(* IEC 61131-3 sources: ics/BLR1_PhoenixContact/BLR1_AXC1050_21/LogicalPOUs/VLV, 3 files *)

(* ---- ValveFB.ST ---- *)
(*@PROPERTIES_EX@
TYPE: POU
LOCALE: 0
IEC_LANGUAGE: ST
PLC_TYPE: independent
PROC_TYPE: independent
GROUP: VLVS.FB
*)
(*@KEY@:DESCRIPTION*)

(*@KEY@:END_DESCRIPTION*)
FUNCTION_BLOCK ValveFB

(*Group:Default*)

VAR
    Fb_Alrm_Tmr :    TON;
END_VAR

VAR_IN_OUT
    Vlv_strct :    VLV;
    Aux_strct :    VLV_MISC;
END_VAR

VAR
    AlrmNotMove :    BOOL;
    AlrmSQ :    BOOL;
    RunManual :    BOOL;
    RunAuto :    BOOL;
    COM_Open :    BOOL;
    COM_Close :    BOOL;
END_VAR

VAR_INPUT
    Cycle :    CCL;
END_VAR

VAR
    NotMove_Alrm_Tmr :    TON;
    AlrmFeedBack :    BOOL;
    AlarmBlock :    BOOL;
END_VAR

VAR_EXTERNAL
    TICK_1S_PLS :    BOOL;
END_VAR

(*@KEY@: WORKSHEET
NAME: ValveFB
IEC_LANGUAGE: ST
*)

IF TICK_1S_PLS and not Aux_strct.AuxFlag THEN
    Aux_strct.Tick_1S:= TRUE;
END_IF;
Aux_strct.AuxFlag:= TICK_1S_PLS;

(*============================================================================*)
    (*Alarm Feedback processing*)
(*============================================================================*)
IF Vlv_strct.CW.Enable and (Aux_strct.COM_Close or Aux_strct.COM_Open) and
    not Vlv_strct.SW.RUN THEN
    IF Aux_strct.Tick_1S THEN
        Aux_strct.FbAlarmTickCount:= Aux_strct.FbAlarmTickCount + 1;
    END_IF;
ELSE
    Aux_strct.FbAlarmTickCount:= 0;
END_IF;

IF Vlv_strct.CW.Enable and ((Aux_strct.COM_Close and not Vlv_strct.SW.Closed) or
    (Aux_strct.COM_Open and not Vlv_strct.SW.Opened)) THEN
    IF Aux_strct.Tick_1S THEN
        Aux_strct.MoveAlarmTickCount:= Aux_strct.MoveAlarmTickCount + 1;
    END_IF;
ELSE
    Aux_strct.MoveAlarmTickCount:= 0;
END_IF;

IF Aux_strct.FbAlarmTickCount >= 3 THEN
    Aux_strct.AlarmFeedBack:= TRUE;
    Aux_strct.FbAlarmTickCount:= 0;
END_IF;

IF Aux_strct.MoveAlarmTickCount >= Aux_strct.SetOvertime THEN
    Aux_strct.AlarmNotMove:= TRUE;
    Aux_strct.MoveAlarmTickCount:= 0;
END_IF;

IF (not Vlv_strct.CW.ExtraEn and (Aux_strct.COM_Open or Aux_strct.COM_Close)) THEN
    Aux_strct.AlarmBlock:= TRUE;
END_IF;

IF Vlv_strct.SW.Opened and Vlv_strct.SW.Closed THEN
    Aux_strct.AlarmSQ:=TRUE;
END_IF;

Vlv_strct.SW.AlarmAccum:= Aux_strct.AlarmNotMove or Aux_strct.AlarmSQ or
    Aux_strct.AlarmFeedBack or Vlv_strct.CW.ExtraAlarm;

IF Vlv_strct.CW.ACK THEN
    Vlv_strct.SW.AlarmAccum:=FALSE;
    Aux_strct.AlarmFeedBack:=FALSE;
    Aux_strct.AlarmSQ:=FALSE;
    Aux_strct.AlarmnotMove:=FALSE;
    Aux_strct.AlarmBlock:= FALSE;
END_IF;

(*============================================================================*)
    (*Auto/Manual mode selection*)
(*============================================================================*)
IF Vlv_strct.CW.AutoMode THEN
    Vlv_strct.SW.ManAuto:= TRUE;
END_IF;
IF Vlv_strct.CW.ManMode THEN
    Vlv_strct.SW.ManAuto:= FALSE;
END_IF;

Vlv_strct.SW.ManOK:=not Vlv_strct.SW.AlarmAccum and Vlv_strct.CW.AuxON and
    Vlv_strct.CW.Enable and not Vlv_strct.SW.ManAuto;

Vlv_strct.SW.AutoOK:= not Vlv_strct.SW.AlarmAccum and Vlv_strct.CW.AuxON and
    Vlv_strct.CW.Enable and Vlv_strct.SW.ManAuto;

(*============================================================================*)
    (*Manual mode activation*)
(*============================================================================*)
IF Vlv_strct.CW.ManOpen or Vlv_strct.CW.ManClose THEN
    Vlv_strct.SW.RunManual:=TRUE;
END_IF;

IF Vlv_strct.CW.Stop or not Vlv_strct.SW.ManOK THEN
    Vlv_strct.SW.RunManual:=FALSE;
END_IF;

(*============================================================================*)
    (*Auto mode activation*)
(*============================================================================*)
Vlv_strct.SW.RunAuto:= Vlv_strct.SW.AutoOK and Cycle.SW.Running;

(*============================================================================*)
    (*Set command for start*)
(*============================================================================*)
Aux_strct.COM_Open:=((Vlv_strct.CW.AutoOpen and Vlv_strct.SW.RunAuto and
    Vlv_strct.SW.AutoOK) or ((Vlv_strct.CW.ManOpen or Aux_strct.COM_Open) and
    Vlv_strct.SW.RunManual and Vlv_strct.SW.ManOK)) and
    not Aux_strct.COM_Close and not Vlv_strct.SW.Opened;

Aux_strct.COM_Close:=((Vlv_strct.CW.AutoClose and Vlv_strct.SW.RunAuto and
    Vlv_strct.SW.AutoOK) or ((Vlv_strct.CW.ManClose or Aux_strct.COM_Close) and
    Vlv_strct.SW.RunManual and Vlv_strct.SW.ManOK)) and
    not Aux_strct.COM_Open and not Vlv_strct.SW.Closed;

Vlv_strct.SW.COM_Open:=Aux_strct.COM_Open and not Vlv_strct.CW.SimEn;
Vlv_strct.SW.COM_Close:=Aux_strct.COM_Close and not Vlv_strct.CW.SimEn;

(*============================================================================*)
    (*Status processing*)
(*============================================================================*)
IF Vlv_strct.SW.AlarmAccum THEN
    Vlv_strct.Status:=word#4;
elsIF not Vlv_strct.CW.ExtraEn THEN
    Vlv_strct.Status:=word#8;
elsIF Vlv_strct.SW.Opened THEN
    Vlv_strct.Status:=word#1;
elsIF Vlv_strct.SW.Closed THEN
    Vlv_strct.Status:=word#2;
ELSE
    Vlv_strct.Status:=word#0;
END_IF;

Vlv_strct.CW.AutoMode:=FALSE;
Vlv_strct.CW.ManMode:=FALSE;
Vlv_strct.CW.ManOpen:=FALSE;
Vlv_strct.CW.Stop:=FALSE;
Vlv_strct.CW.ManClose:=FALSE;
Vlv_strct.CW.ACK:=FALSE;
Aux_strct.Tick_1S:= FALSE;
(*@KEY@: END_WORKSHEET *)
END_FUNCTION_BLOCK

(* ---- VLV.ST ---- *)
(*@PROPERTIES_EX@
TYPE: POU
LOCALE: 0
IEC_LANGUAGE: ST
PLC_TYPE: independent
PROC_TYPE: independent
GROUP: VLVS
*)
(*@KEY@:DESCRIPTION*)

(*@KEY@:END_DESCRIPTION*)
PROGRAM VLV

(*Group:Default*)

VAR_EXTERNAL
    Cycle :CCL;
    V :VALVE;
END_VAR

VAR
    i :INT;
    ValvesFB :ValveFB;
END_VAR

VAR_EXTERNAL
    V_AUX :VALVE_MISC;
END_VAR

VAR
    j :INT;
END_VAR

VAR_EXTERNAL
    MBTCP_Data :MB_TCP_ARR_W_0_7167;
END_VAR

VAR
    VLV_Cycle :CCL;
END_VAR

VAR_EXTERNAL
    AI :SENSOR;
END_VAR

(*@KEY@: WORKSHEET
NAME: VLV
IEC_LANGUAGE: ST
*)
(*============================================================================*)
    (*Valve TV7001 structure parameters*)
(*============================================================================*)
V[0].CW.Enable:= V[0].SW.Rem;
V[0].CW.AuxON:= Cycle.CW.AuxON;
V[0].CW.ExtraEn:= true;
V[0].SW.RUN:= V[0].SW.COM_Open or V[0].SW.COM_Close;
V[0].ActPos:= AI[91].RealValue;
V_AUX[0].SetOvertime:= 180;

(*============================================================================*)
    (*Valve TV8019 structure parameters*)
(*============================================================================*)
V[1].CW.Enable:= V[1].SW.Rem;
V[1].CW.AuxON:= Cycle.CW.AuxON;
V[1].CW.ExtraEn:= true;
V[1].SW.RUN:= V[1].SW.COM_Open or V[1].SW.COM_Close;
V[1].ActPos:= AI[92].RealValue;
V_AUX[1].SetOvertime:= 70;

(*============================================================================*)
    (*Valve TV9008 structure parameters*)
(*============================================================================*)
V[2].CW.Enable:= V[2].SW.Rem;
V[2].CW.AuxON:= Cycle.CW.AuxON;
V[2].CW.ExtraEn:= true;
V[2].SW.RUN:= V[2].SW.COM_Open or V[2].SW.COM_Close;
V[2].ActPos:= AI[93].RealValue;
V_AUX[2].SetOvertime:= 70;

(*============================================================================*)
    (*Valve HV5004 structure parameters*)
(*============================================================================*)
V[3].CW.Enable:= true;
V[3].CW.AuxON:= Cycle.CW.AuxON;
V[3].CW.ExtraEn:= true;
V[3].SW.RUN:= V[3].SW.COM_Open;
V[3].SW.Opened:= V[3].SW.COM_Open;
V_AUX[3].SetOvertime:= 3;

(*============================================================================*)
    (*Valve HV8009 structure parameters*)
(*============================================================================*)
V[4].CW.Enable:= true;
V[4].CW.AuxON:= Cycle.CW.AuxON;
V[4].CW.ExtraEn:= true;
V[4].SW.RUN:= V[4].SW.COM_Open;
V[4].SW.Opened:= V[4].SW.COM_Open;
V_AUX[4].SetOvertime:= 3;

(*============================================================================*)
    (*Valve HV016 structure parameters*)
(*============================================================================*)
V[5].CW.Enable:= true;
V[5].CW.AuxON:= Cycle.CW.AuxON;
V[5].CW.ExtraEn:= true;
V[5].SW.RUN:= V[5].SW.COM_Open;
V[5].SW.Opened:= V[5].SW.COM_Open;
V_AUX[5].SetOvertime:= 3;

(*============================================================================*)
    (*Valve HV017 structure parameters*)
(*============================================================================*)
V[6].CW.Enable:= true;
V[6].CW.AuxON:= Cycle.CW.AuxON;
V[6].CW.ExtraEn:= true;
V[6].SW.RUN:= V[6].SW.COM_Open;
V[6].SW.Opened:= V[6].SW.COM_Open;
V_AUX[6].SetOvertime:= 3;

(*============================================================================*)
    (*Valve HV018 structure parameters*)
(*============================================================================*)
V[7].CW.Enable:= true;
V[7].CW.AuxON:= Cycle.CW.AuxON;
V[7].CW.ExtraEn:= true;
V[7].SW.RUN:= V[7].SW.COM_Open;
V[7].SW.Opened:= V[7].SW.COM_Open;
V_AUX[7].SetOvertime:= 3;

(*============================================================================*)
    (*Valve HV024 structure parameters*)
(*============================================================================*)
V[8].CW.Enable:= true;
V[8].CW.AuxON:= Cycle.CW.AuxON;
V[8].CW.ExtraEn:= true;
V[8].SW.RUN:= V[8].SW.COM_Open;
V[8].SW.Opened:= V[8].SW.COM_Open;
V_AUX[8].SetOvertime:= 3;

(*============================================================================*)
    (*Valves FB processing*)
(*============================================================================*)
for i:= 0 to 8 do
    j:= i * 16 + 4580;
    VLV_Cycle.SW.Running:= V[i].SW.ManAuto;
    ValvesFB(Vlv_strct:=V[i],Aux_strct:=V_AUX[i],Cycle:=VLV_Cycle);
    V[i]:=ValvesFB.Vlv_strct;
    V_AUX[i]:=ValvesFB.Aux_strct;
end_for;

(*============================================================================*)

(*@KEY@: END_WORKSHEET *)
END_PROGRAM

(* ---- VLV_CTRL.ST ---- *)
(*@PROPERTIES_EX@
TYPE: POU
LOCALE: 0
IEC_LANGUAGE: ST
PLC_TYPE: independent
PROC_TYPE: independent
GROUP: VLVS
*)
(*@KEY@:DESCRIPTION*)

(*@KEY@:END_DESCRIPTION*)
PROGRAM VLV_CTRL

(*Group:Default*)

VAR_EXTERNAL
    AI :	SENSOR;
    RGLTR :	REGULATOR;
    V :	VALVE;
END_VAR

VAR
    OP_Req :	BOOL;
    CL_Req :	BOOL;
END_VAR

VAR_EXTERNAL
    TICK_1S_PLS :	BOOL;
END_VAR

VAR
    CNT :	INT;
    PLS_GEN :	BOOL;
    R_TRIG_1 :	R_TRIG;
END_VAR

VAR_EXTERNAL
    TICK_1S :	BOOL;
END_VAR

VAR
    CNT1 :	INT;
    CNT2 :	INT;
    PLS_GEN1 :	BOOL;
    PLS_GEN2 :	BOOL;
    OP_Req1 :	BOOL;
    CL_Req1 :	BOOL;
    OP_Req2 :	BOOL;
    CL_Req2 :	BOOL;
    HW_PID :	FPID;
    HW_SCAN_TMR :	TON;
    HW_SCAN_INIT :	BOOL;
    SW_PID :	FPID;
    SW_SCAN_TMR :	TON;
    SW_SCAN_INIT :	BOOL;
    HC_PID :	FPID;
    HC_SCAN_TMR :	TON;
    HC_SCAN_INIT :	BOOL;
END_VAR

(*@KEY@: WORKSHEET
NAME: VLV_CTRL
IEC_LANGUAGE: ST
*)
(*============================================================================*)
    (*Heat Carier temperature controling*)
(*============================================================================*)
RGLTR[10].CW.En:= V[0].SW.ManAuto;
RGLTR[10].ActVal:= AI[60].RealValue;

HC_PID(REMOTE:=RGLTR[10].CW.En,
        AUTO:=true,
        DIRECTN:=FALSE,
        INTLCK:=FALSE,
        Tscan:=1.0,
        Yman:=RGLTR[10].ManVal,
        SPR:=RGLTR[10].SP,
        SPL:=0.0,X:=RGLTR[10].ActVal,
        KP:=RGLTR[10].Kp,
        TI:=RGLTR[10].Tn,
        TD:=RGLTR[10].Tv,
        HIGH:=100.0,
        LOW:=0.0,
        INTLCKV:=0.0);
RGLTR[10].Y:=HC_PID.Yout;

HC_SCAN_TMR(IN:=not HC_SCAN_TMR.Q and not HC_SCAN_INIT,PT:=t#10S);

IF HC_SCAN_TMR.Q  and not AI[91].SW.Fault and not AI[60].SW.Fault TRUE
    HC_SCAN_INIT:= true;
END_IF;

IF HC_SCAN_INIT TRUE
    V[0].CW.AutoOpen:= (AI[91].RealValue < (RGLTR[10].Y - RGLTR[10].DeadBand)) and not V[0].SW.Opened;
    V[0].CW.AutoClose:= (AI[91].RealValue > (RGLTR[10].Y + RGLTR[10].DeadBand)) and not V[0].SW.Closed;
END_IF;

IF not V[0].CW.AutoOpen and not V[0].CW.AutoClose and HC_SCAN_INIT TRUE
    HC_SCAN_INIT:= FALSE;
END_IF;

(*R_TRIG_1(CLK:=TICK_1S);

IF R_TRIG_1.Q TRUE
    CNT:= CNT + 1;
    CNT1:= CNT1 + 1;
    CNT2:= CNT2 + 1;
END_IF;

IF CNT < 5 TRUE
    PLS_GEN:= true;
elsIF CNT > 185 TRUE
    CNT:= 0;
else
    PLS_GEN:= FALSE;
END_IF;

RGLTR[10].ActVal:= AI[58].RealValue;

OP_Req:= (RGLTR[10].ActVal < (RGLTR[10].SP - (RGLTR[10].DeadBand / 2.0)));
CL_Req:= (RGLTR[10].ActVal > (RGLTR[10].SP + (RGLTR[10].DeadBand / 2.0)));

V[0].CW.AutoOpen:= OP_Req and PLS_GEN;
V[0].CW.AutoClose:= CL_Req and PLS_GEN;*)

(*============================================================================*)
    (*Hot water temperature controling*)
(*============================================================================*)
RGLTR[11].CW.En:= V[1].SW.ManAuto;
RGLTR[11].ActVal:= AI[64].RealValue;

HW_PID(REMOTE:=RGLTR[11].CW.En,
        AUTO:=true,
        DIRECTN:=FALSE,
        INTLCK:=FALSE,
        Tscan:=1.0,
        Yman:=RGLTR[11].ManVal,
        SPR:=RGLTR[11].SP,
        SPL:=0.0,
        X:=RGLTR[11].ActVal,
        KP:=RGLTR[11].Kp,
        TI:=RGLTR[11].Tn,
        TD:=RGLTR[11].Tv,
        HIGH:=100.0,
        LOW:=0.0,
        INTLCKV:=0.0);
RGLTR[11].Y:=HW_PID.Yout;

HW_SCAN_TMR(IN:=not HW_SCAN_TMR.Q and not HW_SCAN_INIT,PT:=t#10S);

IF HW_SCAN_TMR.Q  and not AI[92].SW.Fault and not AI[64].SW.Fault TRUE
    HW_SCAN_INIT:= true;
END_IF;

IF HW_SCAN_INIT TRUE
    V[1].CW.AutoOpen:= (AI[92].RealValue < (RGLTR[11].Y - RGLTR[11].DeadBand)) and
    not V[1].SW.Opened;
    V[1].CW.AutoClose:= (AI[92].RealValue > (RGLTR[11].Y + RGLTR[11].DeadBand)) and
    not V[1].SW.Closed;
END_IF;

IF not V[1].CW.AutoOpen and not V[1].CW.AutoClose and HW_SCAN_INIT TRUE
    HW_SCAN_INIT:= FALSE;
END_IF;

(*
IF CNT1 < 3 TRUE
    PLS_GEN1:= true;
elsIF CNT1 > 30 TRUE
    CNT1:= 0;
else
    PLS_GEN1:= FALSE;
END_IF;

OP_Req1:= (RGLTR[11].ActVal < (RGLTR[11].SP - (RGLTR[11].DeadBand / 2.0)));
CL_Req1:= (RGLTR[11].ActVal > (RGLTR[11].SP + (RGLTR[11].DeadBand / 2.0)));

V[1].CW.AutoOpen:= OP_Req1 and PLS_GEN1;
V[1].CW.AutoClose:= CL_Req1 and PLS_GEN1;*)

(*============================================================================*)
    (*Supply water temperature controling*)
(*============================================================================*)

RGLTR[12].CW.En:= V[2].SW.ManAuto;
RGLTR[12].ActVal:= AI[74].RealValue;

SW_PID(REMOTE:=RGLTR[12].CW.En,
        AUTO:=true,
        DIRECTN:=FALSE,
        INTLCK:=FALSE,
        Tscan:=1.0,
        Yman:=RGLTR[12].ManVal,
        SPR:=RGLTR[12].SP,
        SPL:=0.0,
        X:=RGLTR[12].ActVal,
        KP:=RGLTR[12].Kp,
        TI:=RGLTR[12].Tn,
        TD:=RGLTR[12].Tv,
        HIGH:=100.0,
        LOW:=0.0,
        INTLCKV:=0.0);
RGLTR[12].Y:=SW_PID.Yout;

SW_SCAN_TMR(IN:=not SW_SCAN_TMR.Q and not SW_SCAN_INIT,PT:=t#10S);

IF SW_SCAN_TMR.Q  and not AI[93].SW.Fault and not AI[74].SW.Fault TRUE
    SW_SCAN_INIT:= true;
END_IF;

IF SW_SCAN_INIT TRUE
    V[2].CW.AutoOpen:= (AI[93].RealValue < (RGLTR[12].Y - RGLTR[12].DeadBand)) and
    not V[2].SW.Opened;
    V[2].CW.AutoClose:= (AI[93].RealValue > (RGLTR[12].Y + RGLTR[12].DeadBand)) and
    not V[2].SW.Closed;
END_IF;

IF not V[2].CW.AutoOpen and not V[2].CW.AutoClose and SW_SCAN_INIT TRUE
    SW_SCAN_INIT:= FALSE;
END_IF;

(*
IF CNT2 < 3 TRUE
    PLS_GEN2:= true;
elsIF CNT2 > 60 TRUE
    CNT2:= 0;
else
    PLS_GEN2:= FALSE;
END_IF;

RGLTR[12].ActVal:= AI[72].RealValue;

OP_Req2:= (RGLTR[12].ActVal < (RGLTR[12].SP - (RGLTR[12].DeadBand / 2.0)));
CL_Req2:= (RGLTR[12].ActVal > (RGLTR[12].SP + (RGLTR[12].DeadBand / 2.0)));

V[2].CW.AutoOpen:= OP_Req2 and PLS_GEN2;
V[2].CW.AutoClose:= CL_Req2 and PLS_GEN2;
*)
(*@KEY@: END_WORKSHEET *)
END_PROGRAM
